(* IEC 61131-3 sources: Industry-PLC-LLM/data/PLCBEAD_repo/PLCBEAD_PLCEmbed-main/PLC-BEAD/Source/GEB/BIT_TOGGLE_DW, 1 file *)

(* ---- BIT_TOGGLE_DW.ST ---- *)
FUNCTION BIT_TOGGLE_DW:DWORD
	VAR_INPUT
		IN :	DWORD;
		POS :	INT;
	END_VAR

	BIT_TOGGLE_DW := SHL(DWORD#1, POS) XOR IN;

END_FUNCTION

PROGRAM program0
  VAR
    LocalVar0 : DWORD;
    LocalVaR1  : INT;
    CEIL5_OUT : DWORD;
  END_VAR

  CEIL5_OUT := BIT_TOGGLE_DW(LocalVar0, LocalVaR1 );
END_PROGRAM
